TYPE ActorStartMovingtimeoutEx_t :
STRUCT
	ActorStartMovingTimeout : GernericErrorWatchdog_t;
	expectedActorValue : BOOL; // actor value when sensor is true
	sensorPtr : POINTER TO BOOL := NULL;
	actorPtr : POINTER TO BOOL := NULL;
	sensorID : sensorID_t := sensorID_t.SENSOR_NO_SENSOR;
	actorID : actorID_t := actorID_t.ACTOR_NO_ACTOR;
END_STRUCT
END_TYPE

(* stored: Version 1.1.0.1
   DUT ActorStartMovingtimeoutEx_t: Id {1014532c-e603-403a-958a-a4d249cd9ef6} *)
